INTERFACE Reader EXTENDS __SYSTEM.IQueryInterface

END_INTERFACE

(* stored: Version 1.1.0.1
   Itf Reader: Id {7276acb6-fffb-4468-8690-6aa1c7cbb0f3} *)
